(* CoDeSys 2.3.9.41 project: Котел_розжиг (1).pro *)
(* Libraries: Standard.lib 4.10.05 11:14:46, SYSLIBCALLBACK.LIB 26.9.08 16:43:52, Util.lib 18.5.10 15:14:28, SysLibFile.lib 23.9.04 10:11:36 *)

(* Global variable list: Global_Variables *)
VAR_GLOBAL

	(*Ошибка *)
	Error:BOOL;
	codeError:WORD;

	(*Тригеры*)
	stopTrig: F_TRIG;
	startTrig: F_TRIG;

	(*Уставка воды*)
	tempSpOut:REAL;

	(*state*)
	start:BOOL;
	stop:BOOL;
	gasMode:BOOL;
	oilMode:BOOL;


	(*Датчики *)
	gasConsum:REAL;
	oilConsum:REAL;
	waterInTemp:REAL;
	waterOutTemp:REAL;
	waterOutPressure:REAL;
	waterOutConsum:REAL;
	flameSensor:REAL;
	conceCO2Sensor:REAL;
	oilPressureSensor:REAL;
	gasPressureSensor:REAL;

	(*Блок ошибок*)
	gasConsumError:SensError;
	oilConsumError:SensError;
	waterInTempError:SensError;
	waterOutTempError:SensError;
	waterOutPressureError:SensError;
	waterOutConsumError:SensError;
	flameSensorError:SensError;
	conceCO2SensorError:SensError;

	(*Клапана*)
	valveWaterTempIn:REAL;
	valveWaterTempOut:REAL;
	valveErrorOil:BOOL;
	valveErrorGas:BOOL;
	valveOilIn:REAL;
	valveGasIn:REAL;
	valveStartFlameOil:REAL;
	valveStartFlameGas:REAL;
	valveMainFlameOil:BOOL;
	valveMainFlameGas:BOOL;
	valveAeratorIn:BOOL;
	valveAeratorOut:BOOL;

	(*Вентиляторы*)
	fanFlame:REAL;
	fanOut:REAL;


	(*PID*)
	pidReg:myPid;
	spMinPidOut:WORD;
	spMaxPidOut:WORD;
	pidOffset, pidOffsetOld: WORD;
	(*Таймер*)
	saveParamTimer:TON;
	waterStartTON:TON;
END_VAR

(* Data type *)
TYPE OptionsBoiler :
STRUCT
	gasMode:BOOL;
	oilMode:BOOL;
	start:BOOL;
	stop:BOOL;
END_STRUCT
END_TYPE

(* POU PLC_PRG, ST *)
PROGRAM PLC_PRG
VAR
END_VAR
stopStart();
sensControl();
waterControl();
errorHandle();
END_PROGRAM
ACTION errorHandle:
Error := gasConsumError.errorOut OR
	oilConsumError.errorOut OR
	waterInTempError.errorOut OR
	waterOutTempError.errorOut OR
	waterOutPressureError.errorOut OR
	waterOutConsumError.errorOut OR
	flameSensorError.errorOut OR
	conceCO2SensorError.errorOut ;
END_ACTION
ACTION sensControl:
	gasConsumError(
	value :=  ,
	errorValueMax:=0,
	errorValueMin:=10,
	errorOut => codeError.7
	);
(*_______________________________________________________________*)
	oilConsumError(
	value :=  ,
	errorValueMax:=0,
	errorValueMin:=10,
	errorOut => codeError.0
	);
(*_______________________________________________________________*)
	waterInTempError(
	value :=  ,
	errorValueMax:=0,
	errorValueMin:=10,
	errorOut => codeError.1
	);
(*_______________________________________________________________*)
	waterOutTempError(
	value :=  ,
	errorValueMax:=0,
	errorValueMin:=10,
	errorOut => codeError.2
	);
(*_______________________________________________________________*)
	waterOutPressureError(
	value :=  ,
	errorValueMax:=0,
	errorValueMin:=10,
	errorOut => codeError.3
	);
(*_______________________________________________________________*)
	waterOutConsumError(
	value :=  ,
	errorValueMax:=0,
	errorValueMin:=10,
	errorOut => codeError.4
	);
(*_______________________________________________________________*)
	flameSensorError(
	value :=  ,
	errorValueMax:=0,
	errorValueMin:=10,
	errorOut => codeError.5
	);
(*_______________________________________________________________*)
	conceCO2SensorError(
	value :=  ,
	errorValueMax:=0,
	errorValueMin:=10,
	errorOut => codeError.6
	);
END_ACTION
ACTION stopStart:
startTrig(CLK:=start);
IF startTrig.Q THEN start := TRUE;
stop:=FALSE;
startTrig.CLK :=FALSE;
END_IF

stopTrig(CLK:=stop);
IF stopTrig.Q THEN stop := TRUE;
	start:=FALSE;
	stopTrig.CLK :=FALSE;
 END_IF
END_ACTION
ACTION waterControl:
waterStartTON(IN:= Start, PT:= T#10s);

IF  NOT(waterStartTON.ET = T#0s ) THEN
	valveWaterTempIn := 100;
	valveAeratorIn:= TRUE;
	valveAeratorOut:=TRUE;
	ELSE

	valveWaterTempIn := 0;
	valveAeratorIn:= FALSE;
	valveAeratorOut:=FALSE;
END_IF


IF NOT Error AND NOT stop AND  NOT(waterStartTON.ET = T#0s )    THEN

	IF spMinPidOut>=spMaxPidOut THEN spMaxPidOut:=spMinPidOut+1; END_IF

	IF PidReg.Y<=spMinPidOut THEN
		pidOffset:=spMinPidOut;
		ELSIF PidReg.Y>=spMaxPidOut THEN
			pidOffset:=spMaxPidOut;
			ELSE
				pidOffset:=pidOffsetOld;
	END_IF
	PidReg(
		actual:=waterOutTemp,
		sp:=tempSpOut,
		spShift:=4,
		KP:=10/100,(*Чисто рандом*)
		TN:=10,(*да*)
		TV:=,
		yManual:=0,
		yOffset:=pidOffset,
		yMin:=50,
		yMax:=165,
		manual:= FALSE,(*pid mode*)
		deadZone:=0.25,
		reset:=PidReg.overflow OR  Error AND  stop AND  waterStartTON.ET = T#0s  ,
		(*Выхода*)
		Y=>);

END_IF;
END_ACTION

(* POU saveLoadParamFile, ST *)
PROGRAM saveLoadParamFile
VAR
	file:				DWORD;
	optBoiler:			OptionsBoiler;

	optionSaveFT: F_TRIG;
	loadTON: TON;
	optionsLoadFT: F_TRIG;
	startLoad: BOOL:=TRUE;
END_VAR
loadTON(IN:=startLoad, PT:=T#50ms);
IF loadTON.Q THEN startLoad:=FALSE; END_IF

optionsLoadFT(CLK:= startLoad);


saveParamTimer(IN:= NOT saveParamTimer.Q , PT:=T#10s);

optionSaveFT(CLK:=saveParamTimer.Q);

IF optionSaveFT.Q THEN
	optBoiler.gasMode := gasMode;
	optBoiler.oilMode := oilMode;
	optBoiler.start := start;
	optBoiler.stop := stop;

	file:=SysFileOpen('options', 'w');
	SysFileWrite(file, ADR(optBoiler), SIZEOF(optBoiler));
	SysFileClose(file);
END_IF

IF optionsLoadFT.Q THEN
	file:=SysFileOpen('options', 'r');
	SysFileRead(file, ADR(optBoiler), SIZEOF(optBoiler));
	SysFileClose(file);

	gasMode:= optBoiler.gasMode;
	oilMode:= optBoiler.oilMode;
	start:=optBoiler.start ;
	stop := optBoiler.stop;
END_IF
END_PROGRAM

(* POU Deriv, ST *)
(* function block to approximate the derivative of a value *)
(* to calculate this, always four values are used in order to be as exact as possible *)
FUNCTION_BLOCK Deriv
VAR_INPUT
	in:REAL;		(* input variable *)
	tm:DWORD;		(* time since last call in msec *)
	reset:BOOL;		(* reset: set OUT to zero *)
END_VAR
VAR_OUTPUT
	out:REAL;		(* derivative *)
END_VAR
VAR
	X3,X2,X1:REAL;
	T2,T1:DWORD;
	init:BOOL:=TRUE;
END_VAR
IF init OR reset THEN
	X1:=in;
	X2:=in;
	X3:=in;
	out:=0;
	init:=FALSE;
ELSE
	IF tm>0 THEN
		out:=(3*(in-X3)+X1-X2)/((3*T2+4*T1+3*tm))*1000;
		X3:=X2;
		X2:=X1;
		X1:=in;
		T2:=T1;
		T1:=tm;
	END_IF;
END_IF;
END_FUNCTION_BLOCK

(* POU Integ, ST *)
(* function block to approximate the integral of IN over the time *)
FUNCTION_BLOCK Integ
VAR_INPUT
	in:REAL;				(* input variable *)
	tm:DWORD;				(* time since last call in msec *)
	reset:BOOL;				(* reset: OUT is set to zero and OVERFLOW to false *)
END_VAR
VAR_OUTPUT
	out:REAL;				(* value of the integral *)
	overflow:BOOL:=FALSE;	(* overflow *)
END_VAR
VAR
END_VAR
IF reset THEN
	out:=0;
	overflow:=FALSE;
ELSIF NOT overflow  THEN
	IF 1E38 - in*tm < out OR -1E38 - in*tm > out THEN
		overflow:=TRUE;
	ELSE
		out:=out+in*tm/1000;
	END_IF;
END_IF;
END_FUNCTION_BLOCK

(* POU myPid, ST *)
FUNCTION_BLOCK myPid
VAR_INPUT
	actual:		REAL;	(*Текущее значение*)
	sp:			REAL;	(*Уставка*)
	spShift:	REAL;	(*Сдвиг уставки для уменьшения скорости ПИД на большом диапазоне, если SPShift<DeadZone то выкл*)
	KP:			REAL;	(*Пропорциональный коэффициент*)
	TN:			REAL;	(*Интегральный коэффициент*)
	TV:			REAL;	(*Время интегрирования в *)
	yManual:	REAL;	(*Y равен этому значению когда MANUAL=TRUE*)
	yOffset:	REAL;	(*Смещение выхода на старте*)
	yMin:		REAL;	(*Минимум выхода*)
	yMax:		REAL;	(*Максимум выхода*)
	manual:		BOOL;	(*Y=YManual когда MANUAL=TRUE *)
	reset:		BOOL;	(*Сброс регулятора Y=YOffset*)
	deadZone:	REAL;	(*Ширина зоны нечувствительности*)
END_VAR
VAR_OUTPUT
	Y:				REAL;			(*Выходное значение*)
	limitsActive:	BOOL:=FALSE;	(*Достигнуты лимиты выхода YMin, YMax *)
	overflow:		BOOL:=FALSE;	(*Переполнение интегральной части*)
END_VAR
VAR
	clock:			TON;
	I: 				Integ;
	D: 				Deriv;
	tmDiff: 		DWORD;
	error: 			REAL;
	init: 			BOOL:=TRUE;
END_VAR
IF TN>0 AND KP<> 0 AND (NOT overflow OR reset OR manual) THEN
	sp:=SEL(spShift>DeadZone, sp, SEL(sp-spShift>actual, sp, actual+spShift));
	error := SEL( ABS(sp-actual)<deadZone, sp-actual, 0);			(* Regeldifferenz *)

	IF reset OR init OR manual THEN	(* Reset oder Handbetrieb *)
		I(Reset:=TRUE);
		D(Reset:=TRUE);
		overflow:=FALSE;
		limitsActive:=FALSE;
		IF reset OR init THEN
			Y := yOffset;
			init:=FALSE;
			ELSIF manual THEN
				Y := yManual;
		END_IF
		tmDiff:=0;
		clock(IN:=FALSE);									(* Timer neu starten *)
		clock(PT:=t#1h, IN:=TRUE);
		ELSE
			clock;											(* Timer abfragen *)
			tmDiff:=TIME_TO_DWORD(Clock.ET);				(* Zeitdifferenz seit letztem Aufruf *)
	END_IF;

	IF tmDiff>0 THEN
		clock(IN:=FALSE);									(* Timer neu starten *)
		clock(PT:=t#1h, IN:=TRUE);

		D(IN:=error, TM:=tmDiff, reset:=FALSE);				(* Differential abschätzen *)
		I(IN:=error, TM:=SEL(limitsActive, tmDiff, 0), reset:=FALSE);				(* Integral abschätzen *)

		overflow := I.overflow;
		IF NOT overflow THEN
			Y:=yOffset+KP*(error+I.out/TN+D.out*TV);
			IF Y>1E30 OR Y<-1E30 THEN					(* Overflow steht bevor, darf aber eigentlich nicht passieren *)
				overflow:=TRUE;
			END_IF;

			limitsActive:=FALSE;
			IF yMax>yMin AND Y>=yMax  THEN				(* Stellwert-Obergrenze ьberschritten *)
				limitsActive:=TRUE;
				IF KP<>0 THEN
					I(IN:=(yMax-Y)*TN/KP, TM:=1000, Reset:=FALSE);	(* Integral korrigieren *)
				END_IF
				Y:=yMax;
			END_IF;

			IF yMax>yMin AND Y<=yMin THEN					(* Stellwert-Untergrenze unterschritten *)
				limitsActive:=TRUE;
				IF KP<>0 THEN
					I(IN:=(yMin-Y)*TN/KP, TM:=1000, Reset:=FALSE);	(* Integral korrigieren *)
				END_IF
				Y:=yMin;
			END_IF;
		END_IF;
	END_IF;

END_IF;
END_FUNCTION_BLOCK

(* POU SensError, ST *)
FUNCTION_BLOCK SensError
VAR_INPUT
	value:REAL;
	errorValueMax:REAL;
	errorValueMin:REAL;
END_VAR
VAR_OUTPUT
	errorOut:BOOL;
END_VAR
VAR
END_VAR
IF value > errorValueMax AND value < errorValueMin THEN
	 errorOut := TRUE;
 END_IF
END_FUNCTION_BLOCK

(* Visualisation ignition
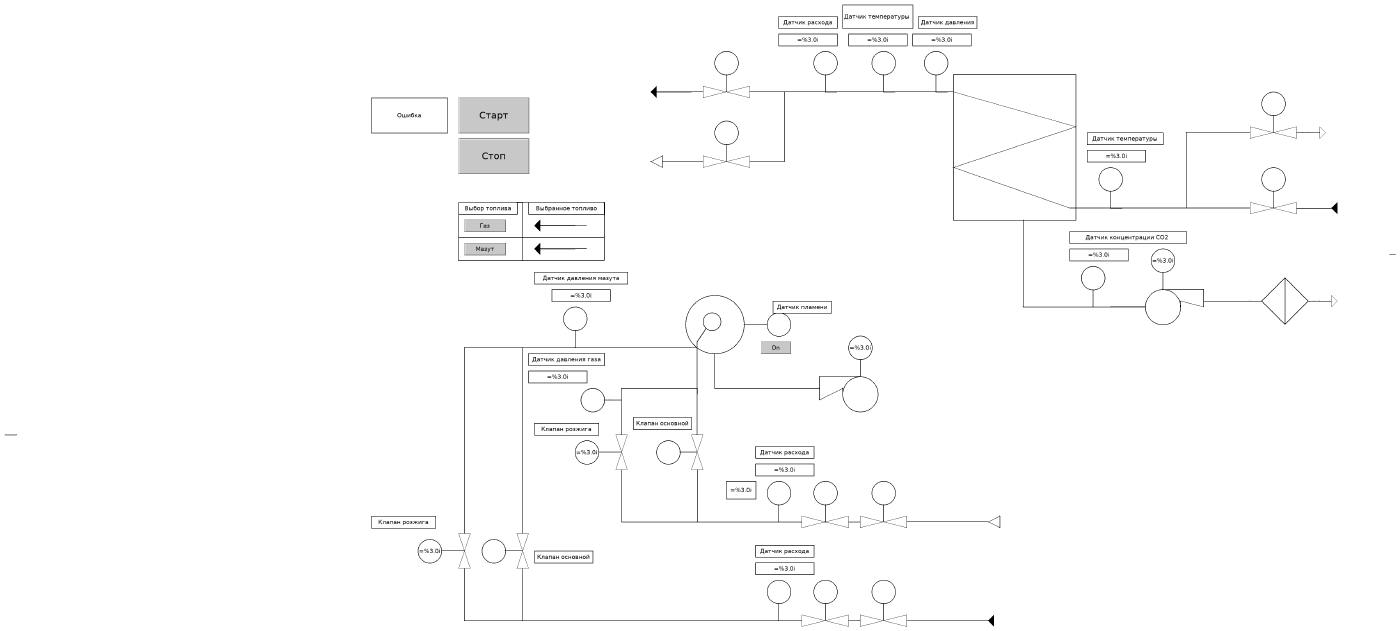
ellipse at (420,740)-(461,781): alarm colour if PLC_PRG.valveNormalFeed
ellipse at (280,740)-(321,781): text "=%3.0i"; shows PLC_PRG.valveLowFeed; alarm colour if PLC_PRG.valveIndicator; editable 0..100
ellipse at (500,520)-(531,551): alarm colour if PLC_PRG.igniter
ellipse at (610,520)-(651,561): alarm colour if PLC_PRG.flameSensor
ellipse at (790,810)-(831,851): alarm colour if PLC_PRG.valveGeneralFeed
rectangle at (590,750)-(691,771): text "Датчик расхода"
rectangle at (210,710)-(321,731): text "Клапан розжига"
rectangle at (380,700)-(481,721): text "Клапан основной"
button at (80,150)-(201,211): text "Старт"; taps start
button at (80,220)-(201,281): text "Стоп"; taps stop
ellipse at (750,560)-(791,601): text "=%3.0i"; shows PLC_PRG.vent; alarm colour if PLC_PRG.ventWork
button at (600,570)-(651,591): text "On"; toggles PLC_PRG.flameButton
rectangle at (590,780)-(691,801): text "=%3.0i"; shows PLC_PRG.fuelSensorLimit; editable 0..1000
rectangle at (540,810)-(591,841): text "=%3.0i"; shows PLC_PRG.consFuelSensor; editable 0..1000
ellipse at (690,810)-(731,851): alarm colour if PLC_PRG.valveAlertStop
ellipse at (1460,270)-(1501,311): alarm colour if PLC_PRG.valveGeneralFeed
ellipse at (520,70)-(561,111): alarm colour if PLC_PRG.valveGeneralFeed
rectangle at (630,10)-(731,31): text "Датчик расхода"
rectangle at (630,40)-(731,61): text "=%3.0i"; shows PLC_PRG.fuelSensorLimit; editable 0..1000
ellipse at (1270,410)-(1311,451): text "=%3.0i"; shows PLC_PRG.vent; alarm colour if PLC_PRG.ventWork
ellipse at (790,980)-(831,1021): alarm colour if PLC_PRG.valveGeneralFeed
rectangle at (590,920)-(691,941): text "Датчик расхода"
rectangle at (590,950)-(691,971): text "=%3.0i"; shows PLC_PRG.fuelSensorLimit; editable 0..1000
ellipse at (690,980)-(731,1021): alarm colour if PLC_PRG.valveAlertStop
ellipse at (120,910)-(161,951): alarm colour if PLC_PRG.valveNormalFeed
ellipse at (10,910)-(51,951): text "=%3.0i"; shows PLC_PRG.valveLowFeed; alarm colour if PLC_PRG.valveIndicator; editable 0..100
rectangle at (-70,870)-(41,891): text "Клапан розжига"
rectangle at (210,930)-(311,951): text "Клапан основной"
ellipse at (520,190)-(561,231): alarm colour if PLC_PRG.valveGeneralFeed
ellipse at (1460,140)-(1501,181): alarm colour if PLC_PRG.valveGeneralFeed
rectangle at (740,-10)-(861,31): text "Датчик температуры"
rectangle at (750,40)-(851,61): text "=%3.0i"; shows PLC_PRG.fuelSensorLimit; editable 0..1000
rectangle at (870,10)-(971,31): text "Датчик давления"
rectangle at (860,40)-(961,61): text "=%3.0i"; shows PLC_PRG.fuelSensorLimit; editable 0..1000
rectangle at (1160,210)-(1291,231): text "Датчик температуры"
rectangle at (1160,240)-(1261,261): text "=%3.0i"; shows PLC_PRG.fuelSensorLimit; editable 0..1000
rectangle at (1130,380)-(1331,401): text "Датчик концентрации CO2"
rectangle at (1130,410)-(1231,431): text "=%3.0i"; shows PLC_PRG.fuelSensorLimit; editable 0..1000
button at (90,360)-(161,381): text "Газ"
button at (90,400)-(161,421): text "Мазут"
rectangle at (620,500)-(721,521): text "Датчик пламени"
rectangle at (620,500)-(721,521): text "Датчик пламени"
rectangle at (80,330)-(181,351): text "Выбор топлива"
rectangle at (200,330)-(331,351): text "Выбранное топливо"
rectangle at (-70,150)-(61,211): text "Ошибка"; alarm colour if Error
rectangle at (210,450)-(371,471): text "Датчик давления мазута"
rectangle at (240,480)-(341,501): text "=%3.0i"; shows PLC_PRG.fuelSensorLimit; editable 0..1000
rectangle at (200,590)-(331,611): text "Датчик давления газа"
rectangle at (200,620)-(301,641): text "=%3.0i"; shows PLC_PRG.fuelSensorLimit; editable 0..1000
90 more shapes without text or variables
*)
